ADAPTER EVENT_HS (* Handshake pattern adapter interface (dataless): CNF/IND in, REQ/RSP out *)
  (* Standard: 61499-1; Description: Copyright (c) 2026 HR Agrartechnik GmbH This program and the accompanying materials are made available under the terms of the Eclipse Public License 2.0 which is available at https://www.eclipse.org/legal/epl-2.0/ SPDX-License-Identifier: EPL-2.0 *)
  (* Version 1.1, 2026-08-31, Franz Höpfinger, HR Agrartechnik GmbH, Swapped EventInputs/EventOutputs so the Plug plays the Requester role (fires REQ/RSP) and the Socket plays the Responder role (fires CNF/IND) - more natural left-to-right layout in the FBNetwork editor *)
  (* Version 1.0, 2026-08-31, Franz Höpfinger, HR Agrartechnik GmbH, Handshake design pattern (IEC 61499 primer course, Module 6, Valeriy Vyatkin), dataless variant as shown on slide 72 - initial version, Socket was the Requester *)
  PACKAGE adapter::events::Handshake;
  (* Documentation:
  Dataless adapter interface implementing the Handshake design pattern (IEC 61499 primer course, Module 6 – Design methods and patterns, Valeriy Vyatkin, Luleå University of Technology / Aalto University, slide 72, category Behavioural).
   Bundles the classical Request/Confirm/Indication/Response service primitives into a single adapter connection, instead of four separate event connections between the two communication partners.
    - REQ – request from Plug to Socket ("please do X")
   - CNF – confirmation from Socket to Plug, answers a REQ ("X done")
   - IND – unsolicited indication from Socket to Plug ("something happened")
   - RSP – response from Plug to Socket, answers an IND ("indication received")
    Plug (Name>>) keeps the declared direction and plays the Requester/client role: it fires REQ/RSP and reacts to CNF/IND. Socket (>>Name) mirrors the direction and plays the Responder/server role: it reacts to REQ/RSP and fires CNF/IND.
   Confirmed against the actual 4diac ECC compiler: it only checks that HS.<Name> is some event declared on the adapter - it does not check whether the direction makes sense at that Socket/Plug side. Get the Sockets/Plugs declaration and the ECC wiring right on purpose; a swapped/self-referential wiring will still validate.
   This is the minimal, dataless variant exactly as shown on slide 72; no payload variables are declared. See test_AX/Meins/DesingPatterns/HandshakePattern/HandshakePattern.md for the full write-up and usage examples.
  *)
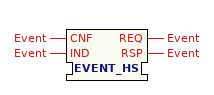
  EVENT_INPUT
    CNF; (* Confirmation from Socket to Plug, answers a REQ *)
    IND; (* Indication from Socket to Plug *)
  END_EVENT
  EVENT_OUTPUT
    REQ; (* Request from Plug to Socket *)
    RSP; (* Response from Plug to Socket, answers an IND *)
  END_EVENT
  SERVICE PLUG/SOCKET
    SEQUENCE request_confirm
      PLUG.REQ() -> SOCKET.REQ();
      SOCKET.CNF() -> PLUG.CNF();
    END_SEQUENCE
    SEQUENCE indication_response
      SOCKET.IND() -> PLUG.IND();
      PLUG.RSP() -> SOCKET.RSP();
    END_SEQUENCE
  END_SERVICE
END_ADAPTER
